VAR_GLOBAL
	xModeStepForStep :BOOL;
    xNextStep :BOOL;
	fbAct1:FB_ActionneurSimple;
END_VAR

(* stored: Version 1.1.0.1, ProductVersion 3.1.4020.6
   GVL GVL: Id {e9ca3882-c39e-4c76-b301-d80faf06cb47} *)
